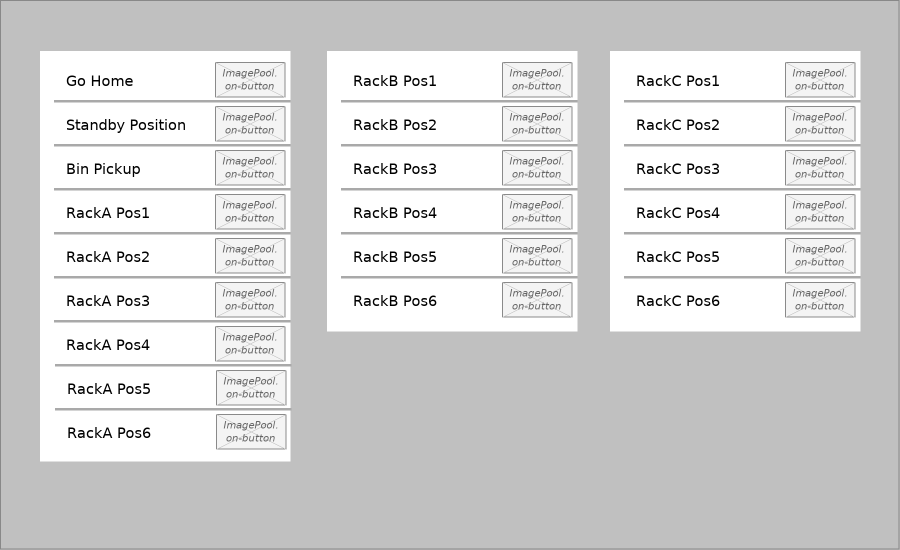
VISUALIZATION KUKA_PROG_CONTENT  // 900x550
    Rectangle (0,0 900x550)
    Group (40,51 251x410)
        RoundedRectangle (0,0 250x410)
        RoundedRectangle (23,21 109x18), "Go Home"
        RoundedRectangle (23,65 125x18), "Standby Position"
        RoundedRectangle (23,109 92x18), "Bin Pickup"
        RoundedRectangle (23,153 92x18), "RackA Pos1"
        RoundedRectangle (23,197 92x18), "RackA Pos2"
        RoundedRectangle (23,241 92x18), "RackA Pos3"
        Rectangle (14,49 236x2)
        Rectangle (14,93 236x2)
        Rectangle (14,137 236x2)
        Rectangle (14,181 236x2)
        Rectangle (14,225 236x2)
        RoundedRectangle (24,373 92x18), "RackA Pos6"
        Rectangle (15,357 236x2)
        RoundedRectangle (23,285 92x18), "RackA Pos4"
        Rectangle (14,269 236x2)
        RoundedRectangle (24,329 92x18), "RackA Pos5"
        Image (175,11 70x35), invisible if: IO_KUKA.bMove_enable, image: ImagePool.off-button
            OnMouseClick: execute { IO_KUKA.bMove_enable := TRUE; }
        Image (175,11 70x35), invisible if: NOT IO_KUKA.bMove_enable, image: ImagePool.on-button
            OnMouseClick: execute { IO_KUKA.bMove_enable := FALSE; }
        Image (175,55 70x35), invisible if: IO_KUKA.bDrive_off, image: ImagePool.off-button
            OnMouseClick: execute { IO_KUKA.bDrive_off := TRUE; }
        Image (175,55 70x35), invisible if: NOT IO_KUKA.bDrive_off, image: ImagePool.on-button
            OnMouseClick: execute { IO_KUKA.bDrive_off := FALSE; }
        Image (175,99 70x35), invisible if: IO_KUKA.bIO_Act, image: ImagePool.off-button
            OnMouseClick: execute { IO_KUKA.bIO_Act := TRUE; }
        Image (175,99 70x35), invisible if: NOT IO_KUKA.bIO_Act, image: ImagePool.on-button
            OnMouseClick: execute { IO_KUKA.bIO_Act := FALSE; }
        Image (175,143 70x35), invisible if: IO_KUKA.bExt_start, image: ImagePool.off-button
            OnMouseClick: execute { IO_KUKA.bExt_start := TRUE; }
        Image (175,143 70x35), invisible if: NOT IO_KUKA.bExt_start, image: ImagePool.on-button
            OnMouseClick: execute { IO_KUKA.bExt_start := FALSE; }
        Image (175,187 70x35), invisible if: IO_KUKA.bConf_msg, image: ImagePool.off-button
            OnMouseClick: execute { IO_KUKA.bConf_msg := TRUE; }
        Image (175,187 70x35), invisible if: NOT IO_KUKA.bConf_msg, image: ImagePool.on-button
            OnMouseClick: execute { IO_KUKA.bConf_msg := FALSE; }
        Image (175,231 70x35), invisible if: IO_KUKA.bDrive_on, image: ImagePool.off-button
            OnMouseClick: execute { IO_KUKA.bDrive_on := TRUE; }
        Image (175,231 70x35), invisible if: NOT IO_KUKA.bDrive_on, image: ImagePool.on-button
            OnMouseClick: execute { IO_KUKA.bDrive_on := FALSE; }
        Image (176,363 70x35), invisible if: IO_KUKA.bDrive_on, image: ImagePool.off-button
            OnMouseClick: execute { IO_KUKA.bDrive_on := TRUE; }
        Image (176,363 70x35), invisible if: NOT IO_KUKA.bDrive_on, image: ImagePool.on-button
            OnMouseClick: execute { IO_KUKA.bDrive_on := FALSE; }
        Image (175,275 70x35), invisible if: IO_KUKA.bDrive_on, image: ImagePool.off-button
            OnMouseClick: execute { IO_KUKA.bDrive_on := TRUE; }
        Image (175,275 70x35), invisible if: NOT IO_KUKA.bDrive_on, image: ImagePool.on-button
            OnMouseClick: execute { IO_KUKA.bDrive_on := FALSE; }
        Image (176,319 70x35), invisible if: IO_KUKA.bDrive_on, image: ImagePool.off-button
            OnMouseClick: execute { IO_KUKA.bDrive_on := TRUE; }
        Image (176,319 70x35), invisible if: NOT IO_KUKA.bDrive_on, image: ImagePool.on-button
            OnMouseClick: execute { IO_KUKA.bDrive_on := FALSE; }
        Rectangle (15,313 236x2)
    Group (327,51 250x280)
        RoundedRectangle (0,0 250x280)
        RoundedRectangle (23,21 109x18), "RackB Pos1"
        RoundedRectangle (23,65 92x18), "RackB Pos2"
        RoundedRectangle (23,109 92x18), "RackB Pos3"
        RoundedRectangle (23,153 92x18), "RackB Pos4"
        RoundedRectangle (23,197 92x18), "RackB Pos5"
        RoundedRectangle (23,241 92x18), "RackB Pos6"
        Image (175,11 70x35), invisible if: IO_KUKA.bMove_enable, image: ImagePool.off-button
            OnMouseClick: execute { IO_KUKA.bMove_enable := TRUE; }
        Image (175,11 70x35), invisible if: NOT IO_KUKA.bMove_enable, image: ImagePool.on-button
            OnMouseClick: execute { IO_KUKA.bMove_enable := FALSE; }
        Image (175,55 70x35), invisible if: IO_KUKA.bDrive_off, image: ImagePool.off-button
            OnMouseClick: execute { IO_KUKA.bDrive_off := TRUE; }
        Image (175,55 70x35), invisible if: NOT IO_KUKA.bDrive_off, image: ImagePool.on-button
            OnMouseClick: execute { IO_KUKA.bDrive_off := FALSE; }
        Image (175,99 70x35), invisible if: IO_KUKA.bIO_Act, image: ImagePool.off-button
            OnMouseClick: execute { IO_KUKA.bIO_Act := TRUE; }
        Image (175,99 70x35), invisible if: NOT IO_KUKA.bIO_Act, image: ImagePool.on-button
            OnMouseClick: execute { IO_KUKA.bIO_Act := FALSE; }
        Image (175,143 70x35), invisible if: IO_KUKA.bExt_start, image: ImagePool.off-button
            OnMouseClick: execute { IO_KUKA.bExt_start := TRUE; }
        Image (175,143 70x35), invisible if: NOT IO_KUKA.bExt_start, image: ImagePool.on-button
            OnMouseClick: execute { IO_KUKA.bExt_start := FALSE; }
        Image (175,187 70x35), invisible if: IO_KUKA.bConf_msg, image: ImagePool.off-button
            OnMouseClick: execute { IO_KUKA.bConf_msg := TRUE; }
        Image (175,187 70x35), invisible if: NOT IO_KUKA.bConf_msg, image: ImagePool.on-button
            OnMouseClick: execute { IO_KUKA.bConf_msg := FALSE; }
        Image (175,231 70x35), invisible if: IO_KUKA.bDrive_on, image: ImagePool.off-button
            OnMouseClick: execute { IO_KUKA.bDrive_on := TRUE; }
        Image (175,231 70x35), invisible if: NOT IO_KUKA.bDrive_on, image: ImagePool.on-button
            OnMouseClick: execute { IO_KUKA.bDrive_on := FALSE; }
        Rectangle (14,49 236x2)
        Rectangle (14,93 236x2)
        Rectangle (14,137 236x2)
        Rectangle (14,181 236x2)
        Rectangle (14,225 236x2)
    Group (610,51 250x280)
        RoundedRectangle (0,0 250x280)
        RoundedRectangle (23,21 109x18), "RackC Pos1"
        RoundedRectangle (23,65 92x18), "RackC Pos2"
        RoundedRectangle (23,109 92x18), "RackC Pos3"
        RoundedRectangle (23,153 92x18), "RackC Pos4"
        RoundedRectangle (23,197 92x18), "RackC Pos5"
        RoundedRectangle (23,241 92x18), "RackC Pos6"
        Image (175,11 70x35), invisible if: IO_KUKA.bMove_enable, image: ImagePool.off-button
            OnMouseClick: execute { IO_KUKA.bMove_enable := TRUE; }
        Image (175,11 70x35), invisible if: NOT IO_KUKA.bMove_enable, image: ImagePool.on-button
            OnMouseClick: execute { IO_KUKA.bMove_enable := FALSE; }
        Image (175,55 70x35), invisible if: IO_KUKA.bDrive_off, image: ImagePool.off-button
            OnMouseClick: execute { IO_KUKA.bDrive_off := TRUE; }
        Image (175,55 70x35), invisible if: NOT IO_KUKA.bDrive_off, image: ImagePool.on-button
            OnMouseClick: execute { IO_KUKA.bDrive_off := FALSE; }
        Image (175,99 70x35), invisible if: IO_KUKA.bIO_Act, image: ImagePool.off-button
            OnMouseClick: execute { IO_KUKA.bIO_Act := TRUE; }
        Image (175,99 70x35), invisible if: NOT IO_KUKA.bIO_Act, image: ImagePool.on-button
            OnMouseClick: execute { IO_KUKA.bIO_Act := FALSE; }
        Image (175,143 70x35), invisible if: IO_KUKA.bExt_start, image: ImagePool.off-button
            OnMouseClick: execute { IO_KUKA.bExt_start := TRUE; }
        Image (175,143 70x35), invisible if: NOT IO_KUKA.bExt_start, image: ImagePool.on-button
            OnMouseClick: execute { IO_KUKA.bExt_start := FALSE; }
        Image (175,187 70x35), invisible if: IO_KUKA.bConf_msg, image: ImagePool.off-button
            OnMouseClick: execute { IO_KUKA.bConf_msg := TRUE; }
        Image (175,187 70x35), invisible if: NOT IO_KUKA.bConf_msg, image: ImagePool.on-button
            OnMouseClick: execute { IO_KUKA.bConf_msg := FALSE; }
        Image (175,231 70x35), invisible if: IO_KUKA.bDrive_on, image: ImagePool.off-button
            OnMouseClick: execute { IO_KUKA.bDrive_on := TRUE; }
        Image (175,231 70x35), invisible if: NOT IO_KUKA.bDrive_on, image: ImagePool.on-button
            OnMouseClick: execute { IO_KUKA.bDrive_on := FALSE; }
        Rectangle (14,49 236x2)
        Rectangle (14,93 236x2)
        Rectangle (14,137 236x2)
        Rectangle (14,181 236x2)
        Rectangle (14,225 236x2)
END_VISUALIZATION

(* stored: Version 1.1.0.1, ProductVersion 3.1.4024.12
   Visu KUKA_PROG_CONTENT: Id {2762981c-7435-49a0-a101-5e4bd6cefa4f} *)
